// TIA Portal V21 export
TYPE "coneCrusherCmd"
   STRUCT
      cmdWord : Word;
   END_STRUCT;
END_TYPE
